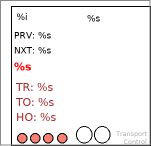
VISUALIZATION V_TransportControl  // 151x146
VAR_IN_OUT	
	{attribute 'VAR_IN_OUT_AS_POINTER'}
	TransportControl	: FB_ProBoxTransportControl;
	ZoneData			: ST_ZoneData;
		
END_VAR
    Rectangle (11,6 140x140), colour toggle: ZoneData.TransportControlData.NumberOfPresentTUs>0
    Rectangle (13,110 130x15), "HO: %s", text variable: ZoneData.TransportControlData.eHandOverState
    Rectangle (13,95 130x15), "TO: %s", text variable: ZoneData.TransportControlData.eTakeOverState
    Rectangle (13,80 130x15), "TR: %s", text variable: ZoneData.TransportControlData.eTransportState
    Rectangle (36,6 115x25), "%s", tooltip "TU ID", text variable: TU_DataTable[ZoneData.TransportControlData.TU_DataIndex].TU_ID.ASCII
    Rectangle (11,28 140x15), "PRV: %s", text variable: TransportControl.PrevTransportData.eFunctionNumber
    Rectangle (11,43 140x15), "NXT: %s", text variable: TransportControl.NextTransportData.eFunctionNumber
    Ellipse (17,133 10x10), tooltip "'Indicator shows that addon(s) is available -> Enable signal'", colour toggle: ZoneData.AddOn.Orders.Enable, invisible if: ZoneData.AddOn.NoAddons
    Ellipse (30,133 10x10), tooltip "'Indicator shows that addon(s) is available - Enable Takeover'", colour toggle: ZoneData.AddOn.Orders.EnableTakeover, invisible if: ZoneData.AddOn.NoAddons
    Ellipse (43,133 10x10), tooltip "'Indicator shows that addon(s) is available - Enable Handover'", colour toggle: ZoneData.AddOn.Orders.EnableHandover, invisible if: ZoneData.AddOn.NoAddons
    Ellipse (57,133 10x10), tooltip "'Indicator shows that addon(s) is available - Data Ready'", colour toggle: ZoneData.AddOn.Orders.DataReady, invisible if: ZoneData.AddOn.NoAddons
    Ellipse (94,126 16x17), tooltip "sensor occupied", colour toggle: ZoneData.TransportControlData.SensorOccupied
    Label (102,130 48x16), "Transport Control"
    Rectangle (11,57 140x20), "%s", tooltip "%s", text variable: ZoneData.ErrorData.Error.ErrorCode.Conv, invisible if: ZoneData.ErrorData.Error.ErrorCode.Conv = 0
        p4168582468: ZoneData.ErrorData.Error.ErrorParam
    Rectangle (11,6 22x22), "%i", tooltip "TU index", text variable: ZoneData.TransportControlData.TU_DataIndex
    Ellipse (76,126 16x17), tooltip "Transportcontrol Occupied", colour toggle: ZoneData.TransportControlData.Occupied
END_VISUALIZATION

(* stored: Version 1.1.0.1, ProductVersion 3.1.4024.9
   Visu V_TransportControl: Id {da3e1b7e-95c2-49bf-970e-9cb62fa3a5da} *)
